// Mitsubishi GX Works2 project: GX W2 L5 Ex 1 DK C   PLC: FX3G

// task Task_01 (event TRUE, interval 0, priority 31): POU_01

PROGRAM POU_01
Y1 := (X1 OR Y1) AND X002;  (* When X1 is On and X2 is On, Y1 is On and Held On *)
Y2 := X003 AND X004;    (* When X3 is On and X4 is On, Y2 is On and Held On *)
Y3 := X3 AND X5;     (*  When X3 is On and X5 is On, Y3 is On and Held On *)
Y4 := (X6 OR Y004) AND NOT X001;   (* When X0 is turned On and Not X1, Y0 switches On and is held On due to Hold-On Contact *)
END_PROGRAM
